// TIA Portal V17 export
// export: Created 2025-06-26T07:49:51.1187588Z, ExportSetting WithDefaults, DisplayName Totally Integrated Automation Portal, DisplayVersion V17 Update 8, DisplayName TIA Portal Openness, DisplayVersion V17 Update 8, DisplayName TIA Portal Version Control Interface, DisplayVersion V17, DisplayName STEP 7 Professional, DisplayVersion V17 Update 8, DisplayName STEP 7 Safety, DisplayVersion V17 Update 6, DisplayName WinCC Advanced, DisplayVersion V17 Update 8
DATA_BLOCK "DB_System"   // DB42
{ S7_Optimized_Access := 'TRUE' }
AUTHOR : Heaten
VERSION : 0.1
// stored: AutoNumber true, DBAccessibleFromOPCUA true, DBAccessibleFromWebserver true, IsOnlyStoredInLoadMemory false, IsRetainMemResEnabled false, IsWriteProtectedInAS false, MemoryReserve 100
   VAR
      bFirstCycle : Bool := FALSE;   // High on first scan only
      bFirstCycleCyclic : Bool := FALSE;
      bSimulation : Bool := FALSE;   // Simulation active
      bProfiling : Bool := FALSE;   // Profiling active
      bInternalEmergencyStop : Bool := FALSE;   // PLC source E-stop. 0 = ok, 1 = Emergency stop
      bExternalEmergencyStop : Bool := FALSE;   // External source E-stop. 0 = ok, 1 = Emergency stop
      bEmergencyStop : Bool := FALSE;   // Emergency stop state. 0 = ok, 1 = Emergency stop
      bManualModeWarning : Bool := FALSE;   // 1 = one or more regulators in manual mode, 0 = no regulators in manual mode
      bExternalValidData { S7_SetPoint := 'True'} : Bool := TRUE;   // 1 = values sent from APP PLC are valid
      fCycleTime : Real := 0.1000159;   // Cycle time in sec
      lfCycleTime : LReal := 0.100015944;   // Cycle time in sec
      BarometricOffset : Real := 101.325;   // [kPa] Pressure offset relative to absolute
   END_VAR
   VAR RETAIN
      SystemUptime : "stHoursCounter";   // System powered on
      SystemActiveTime { S7_SetPoint := 'True'} : "stHoursCounter";   // Standby or higher
      RunningTime { S7_SetPoint := 'True'} : "stHoursCounter";   // In running state
   END_VAR
   VAR
      SafetyRelay { S7_SetPoint := 'True'} : "stSafetyRelay";   // Emergency stop safety relay
      WinCCLink { S7_SetPoint := 'True'} : "stHeartbeat";
   END_VAR
   VAR RETAIN
      AppPLCLink { S7_SetPoint := 'True'} : "stHeartbeatCount2";
   END_VAR
   VAR
      SoftwareVersion : String := 'V4.0.0.6';   // PLC software version string (set in FC35)
   END_VAR
BEGIN
   SystemUptime.nHours := 5956;
   SystemUptime.nMinutes := 7;
   SystemUptime.nSeconds := 43;
   SystemUptime.bReset := FALSE;
   SystemActiveTime.nHours := 0;
   SystemActiveTime.nMinutes := 0;
   SystemActiveTime.nSeconds := 0;
   SystemActiveTime.bReset := FALSE;
   RunningTime.nHours := 0;
   RunningTime.nMinutes := 0;
   RunningTime.nSeconds := 0;
   RunningTime.bReset := FALSE;
   SafetyRelay.tResetLoopTime := T#1S;
   SafetyRelay.tResetTimeout := T#1S;
   SafetyRelay.nState := 3;
   SafetyRelay.bStatus := TRUE;
   SafetyRelay.bResetReq := FALSE;
   SafetyRelay.bResetLoop := FALSE;
   SafetyRelay.bResetCmd := FALSE;
   SafetyRelay.bResetFailed := FALSE;
   WinCCLink.bOut := FALSE;
   WinCCLink.bIn := TRUE;
   WinCCLink.bEnable := TRUE;
   WinCCLink.bOk := TRUE;
   WinCCLink.nState := 2;
   WinCCLink.tTimeout := T#1M_30S;
   AppPLCLink.nLocalCount := 0;
   AppPLCLink.nRemoteCount := 35505;
   AppPLCLink.bEnable := TRUE;
   AppPLCLink.bOk := TRUE;
   AppPLCLink.nState := 2;
   AppPLCLink.tTimeout := T#2S;
END_DATA_BLOCK
